// TIA Portal V20 export
DATA_BLOCK "Global_DB"   // DB16
{ S7_Optimized_Access := 'TRUE' }
// stored: MemoryReserve 100
   VAR
      Auto : Bool;
      Manual : Bool;
      Maintenance : Bool;
      Alarm : Word;
   END_VAR
BEGIN
END_DATA_BLOCK
